// TIA Portal V16 export
// export: Created 2021-04-11T09:51:24.5358486Z, ExportSetting WithDefaults, DisplayName Totally Integrated Automation Portal, DisplayVersion V16, DisplayName TIA Portal Version Control Interface, DisplayVersion V16, DisplayName TIA Portal Openness, DisplayVersion V16, DisplayName STEP 7 Professional, DisplayVersion V16, DisplayName STEP 7 Safety, DisplayVersion V16, DisplayName WinCC Unified SCADA Engineering System, DisplayVersion V16
FUNCTION_BLOCK "preWork_AM"   // FB5, LAD
{ S7_Optimized_Access := 'TRUE' }
VERSION : 0.1
// stored: AutoNumber true, IsIECCheckEnabled false, IsRetainMemResEnabled false, MemoryReserve 100, SetENOAutomatically false, UDAEnableTagReadback false
   VAR_INPUT
      enPreWorkStart : Bool;   // начало пред подготовки
   END_VAR
   VAR_IN_OUT
      alarmStop { ExternalAccessible := 'False'; ExternalVisible := 'False'; ExternalWritable := 'False'} : Bool;   // если пришел аварийный останов
      leftBunker : Array[0..12] of Bool;   // массив закрыть левые бункеры
      rightBunker : Array[0..12] of Bool;   // массив закрыть правые бункеры
      isFinishPreWork : Bool;   // сигнал о окончании подготовки автоматического режима
   END_VAR
   VAR
      closeLeftBunker_FB : Array[0..12] of "controlValve";
      closeRightBunker_FB : Array[0..12] of "controlValve";
      tempButtonLeft : Array[0..12] of Bool;
      tempButtonRight : Array[0..12] of Bool;
      valueControlBit : Bool;
      watchQ : Bool;
      tmpControlValue : Bool;
      tempP_trig : Array[0..1] of Bool;
   END_VAR
   VAR_TEMP
      i : DInt;
   END_VAR
   VAR_TEMP   // added for the SCL form of the ladder/FBD networks
      _w1 : Bool;
      _w2 : Bool;
   END_VAR
BEGIN

REGION Network 1
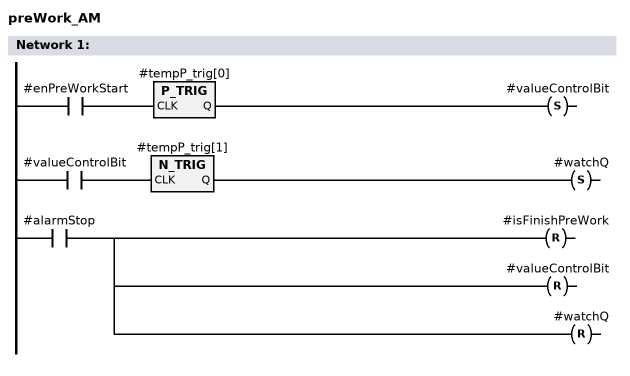
   RUNG wire#powerrail
      Contact( #enPreWorkStart )
      P_Trig( #tempP_trig[0] )
      S_Coil( #valueControlBit )
   END_RUNG
   RUNG wire#powerrail
      Contact( #valueControlBit )
      N_Trig( #tempP_trig[1] )
      S_Coil( #watchQ )
   END_RUNG
   RUNG wire#powerrail
      Contact( #alarmStop )
      wire#w1
      R_Coil( #isFinishPreWork )
   END_RUNG
   RUNG wire#w1
      R_Coil( #valueControlBit )
   END_RUNG
   RUNG wire#w1
      R_Coil( #watchQ )
   END_RUNG
   // the same network as SCL:
   #_w1 := #enPreWorkStart AND NOT #tempP_trig[0];   // rising edge
   #tempP_trig[0] := #enPreWorkStart;
   IF #_w1 THEN #valueControlBit := TRUE; END_IF;
   #_w2 := NOT #valueControlBit AND #tempP_trig[1];   // falling edge
   #tempP_trig[1] := #valueControlBit;
   IF #_w2 THEN #watchQ := TRUE; END_IF;
   IF #alarmStop THEN
       #isFinishPreWork := FALSE;
       #valueControlBit := FALSE;
       #watchQ := FALSE;
   END_IF;
END_REGION

REGION Network 2 (SCL)
       //если нет допуска то нет и разрешения на проверку
       //
       IF NOT (#enPreWorkStart) THEN
           #valueControlBit := false;
           #watchQ := false;
           #isFinishPreWork := false;
       END_IF;

       //проверка(выдержка) пока все закроются
       IF #watchQ THEN
           #i := 0;
           #tmpControlValue := true;
           FOR #i := 1 TO 12 DO
               #tmpControlValue := #tmpControlValue AND NOT (#closeLeftBunker_FB[#i].closeQ);
               #tmpControlValue := #tmpControlValue AND NOT (#closeRightBunker_FB[#i].closeQ);
           END_FOR;
           IF #tmpControlValue THEN//как только все закрыто то проверка закончена
               #watchQ := false;
               #isFinishPreWork := true;
           END_IF;
       END_IF;


       //управление механизмом закрытия
       IF NOT(#isFinishPreWork) THEN
           #i := 0;
           FOR #i := 1 TO 12 DO
               #tempButtonLeft[#i] :=#tempButtonRight[#i] := #valueControlBit;
               #closeLeftBunker_FB[#i](closeQ => #leftBunker[#i],
                                       close := #tempButtonLeft[#i],
                                       stopAlarm := #alarmStop,
                                       "time_open/close":=t#200ms);

               #closeRightBunker_FB[#i](closeQ => #rightBunker[#i],
                                        close := #tempButtonRight[#i],
                                        stopAlarm := #alarmStop,
                                        "time_open/close":=t#200ms);
           END_FOR;
           IF #valueControlBit THEN//сбрасываем бит на закрытие
               #valueControlBit := false;
           END_IF;
       END_IF;
END_REGION
END_FUNCTION_BLOCK
